FUNCTION choldc1 : INT
VAR_IN_OUT
	a:ARRAY[*,*] OF LREAL;
	p:ARRAY[*,*] OF LREAL;
	
END_VAR
VAR_INPUT
	n:SINT;
END_VAR
VAR
	i,j,k:INT;
 	sum:LREAL;
END_VAR

FOR i := 0 TO n DO
            FOR j := i TO n DO
              sum := a[i,j];
              FOR k := i - 1 TO -1 BY -1 DO
                sum := sum - a[i,k] * a[j,k];
	      	  END_FOR
              IF (i = j) THEN
                IF (sum <= 0) THEN
                  choldc1:=1;
				  END_IF
		
                p[i,0] := SQRT(sum);
	     
              ELSE 
                a[j,i] := sum / p[i,0];
	      END_IF
	    END_FOR
	  END_FOR
    choldc1:=0;

END_FUNCTION

(* stored: Version 1.1.0.1, ProductVersion 3.1.4024.12
   POU choldc1: Id {09c7d2dd-ef62-42d8-8ee6-280135f652d6}, SpecialFunc None *)
